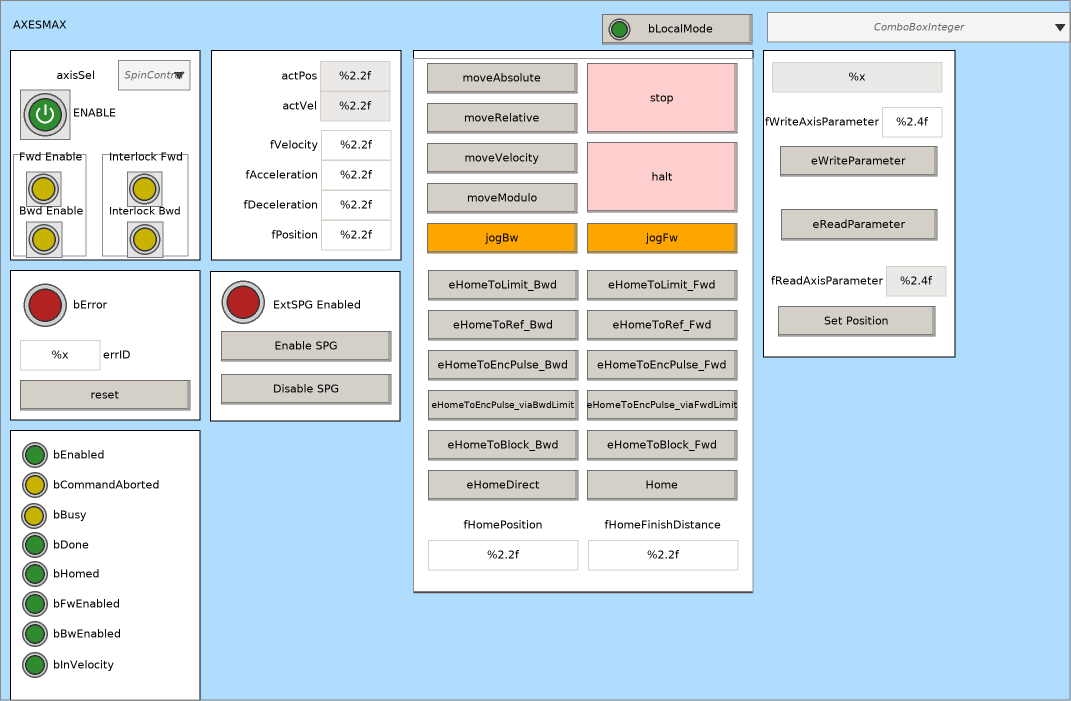
VISUALIZATION MainVisu  // 1071x701
    Rectangle (210,271 190x150)
    Rectangle (413,50 340x542)
    GroupBox (413,50 340x543)
        Button (174,92 150x70), "halt", pressed state: GVL.astAxes[Main.hmiAxisSelection].stControl.bHalt, text list: "languageSupport", text index: "halt"
            toggle GVL.astAxes[Main.hmiAxisSelection].stControl.bHalt
        Button (174,420 150x30), "Home", text list: 'languageSupport', text index: "Home"
            OnMouseClick: execute { GVL.astAxes[Main.hmiAxisSelection].stControl.eCommand:=E_MotionFunctions.eHome; GVL.astAxes[Main.hmiAxisSelection].stControl.bExecute:=TRUE; }
        Button (15,380 150x30), "eHomeToBlock_Bwd", text list: 'languageSupport', text index: "eHomeToBlock_Bwd"
            OnMouseClick: execute {
                GVL.astAxes[Main.hmiAxisSelection].stControl.eCommand:=E_MotionFunctions.eHome;
                GVL.astAxes[Main.hmiAxisSelection].stHomingConfig.eHomeSeq:=E_HomingRoutines.eHomeToBlock_Bwd;
                GVL.astAxes[Main.hmiAxisSelection].stControl.bExecute:=TRUE;
            }
    GroupBox (10,50 190x210)
        Rectangle (0,0 190x210)
        GroupBox (3,96 73x110)
        GroupBox (92,96 86x110)
        Textfield (60,50 92x26), "ENABLE", text list: 'languageSupport', text index: "enable"
        PushSwitchLed (16,118 35x42), variable: GVL.astAxes[MAIN.hmiAxisSelection].stInputs.bLimitFwd, behaviour: TOGGLE, style: Switch-PushSwitchLed-Yellow
        PushSwitchLed (16,170 36x39), variable: GVL.astAxes[MAIN.hmiAxisSelection].stInputs.bLimitBwd, behaviour: TOGGLE, style: Switch-PushSwitchLed-Yellow
        SpinControl (108,10 72x30), variable: MAIN.hmiAxisSelection
            p651134158: GVL_APP.nAXIS_NUM
        Textfield (23,13 86x25), "axisSel", text variable: GVL_APP.nAXIS_NUM, text list: "languageSupport", text index: "axisSel"
        PowerSwitch (10,38 50x53), variable: GVL.astAxes[MAIN.hmiAxisSelection].stControl.bEnable, behaviour: TOGGLE, style: Switch-PowerSwitch-Green
        PushSwitchLed (117,118 35x42), variable: GVL.astAxes[MAIN.hmiAxisSelection].stControl.bInterlockFwd, behaviour: TOGGLE, style: Switch-PushSwitchLed-Yellow
        PushSwitchLed (117,170 36x39), variable: GVL.astAxes[MAIN.hmiAxisSelection].stControl.bInterlockBwd, behaviour: TOGGLE, style: Switch-PushSwitchLed-Yellow
        Textfield (6,94 76x26), "Fwd Enable", text list: 'languageSupport', text index: "enFW"
        Textfield (6,148 76x26), "Bwd Enable", text list: 'languageSupport', text index: "enBW"
        Textfield (96,94 76x26), "Interlock Fwd", text list: 'languageSupport', text index: "bAxisInterlockFwd"
        Textfield (96,148 76x26), "Interlock Bwd", text list: 'languageSupport', text index: "bAxisInterlockBwd"
    Textfield (10,10 231x30), "AXESMAX", text variable: GVL_APP.nAXIS_NUM, text list: "languageSupport", text index: "axesAvailable"
    Button (427,63 150x30), "moveAbsolute", text list: "languageSupport", text index: "moveAbsolute"
        OnMouseClick: execute { GVL.astAxes[MAIN.hmiAxisSelection].stControl.eCommand:=E_MotionFunctions.eMoveAbsolute; GVL.astAxes[MAIN.hmiAxisSelection].stControl.bExecute:=TRUE; }
    Button (427,143 150x30), "moveVelocity", text list: "languageSupport", text index: "moveVelocity"
        OnMouseClick: execute { GVL.astAxes[Main.hmiAxisSelection].stControl.eCommand:=E_MotionFunctions.eMoveVelocity; GVL.astAxes[Main.hmiAxisSelection].stControl.bExecute:=TRUE; }
    Button (427,103 150x30), "moveRelative", text list: "languageSupport", text index: "moveRelative"
        OnMouseClick: execute { GVL.astAxes[Main.hmiAxisSelection].stControl.eCommand:=E_MotionFunctions.eMoveRelative; GVL.astAxes[Main.hmiAxisSelection].stControl.bExecute:=TRUE; }
    Button (427,183 150x30), "moveModulo", text list: "languageSupport", text index: "moveModulo"
        OnMouseClick: execute { GVL.astAxes[Main.hmiAxisSelection].stControl.eCommand:=E_MotionFunctions.eMoveModulo; GVL.astAxes[Main.hmiAxisSelection].stControl.bExecute:=TRUE; }
    Button (587,63 150x70), "stop", pressed state: GVL.astAxes[Main.hmiAxisSelection].stControl.bStop, text list: "languageSupport", text index: "stop"
        toggle GVL.astAxes[Main.hmiAxisSelection].stControl.bStop
    Button (427,223 150x30), "jogBw", text list: "languageSupport", text index: "jogBw"
        OnMouseDown: execute {
            GVL.astAxes[Main.hmiAxisSelection].stControl.eCommand:=E_MotionFunctions.eMoveVelocity;
            GVL.astAxes[Main.hmiAxisSelection].stControl.fVelocity:=-ABS(GVL.astAxes[Main.hmiAxisSelection].stControl.fJogVelocity)
            GVL.astAxes[Main.hmiAxisSelection].stControl.bExecute:= TRUE;
        }
        OnMouseClick: execute {  }
        OnMouseUp: execute { GVL.astAxes[Main.hmiAxisSelection].stControl.bHalt:= TRUE; }
    Button (587,223 150x30), "jogFw", text list: "languageSupport", text index: "jogFw"
        OnMouseDown: execute {
            GVL.astAxes[Main.hmiAxisSelection].stControl.eCommand:=E_MotionFunctions.eMoveVelocity;
            GVL.astAxes[Main.hmiAxisSelection].stControl.fVelocity:=ABS(GVL.astAxes[Main.hmiAxisSelection].stControl.fJogVelocity)
            GVL.astAxes[Main.hmiAxisSelection].stControl.bExecute:= TRUE;
        }
        OnMouseClick: execute {  }
        OnMouseUp: execute { GVL.astAxes[Main.hmiAxisSelection].stControl.bHalt:= TRUE; }
    GroupBox (10,270 190x150)
        Rectangle (0,0 190x150)
        Textfield (90,70 90x30), "errID", text list: "languageSupport", text index: "errID"
        Textfield (10,70 80x30), "%x", text variable: GVL.astAxes[MAIN.hmiAxisSelection].stStatus.nErrorID
        Lamp1 (10,10 50x50), variable: GVL.astAxes[MAIN.hmiAxisSelection].stStatus.bError, style: Lamp-Lamp1-Red
        Textfield (60,20 120x30), "bError", text list: "languageSupport", text index: "bError"
        Button (10,110 170x30), "reset", pressed state: GVL.astAxes[Main.hmiAxisSelection].stControl.bReset, text list: "languageSupport", text index: "reset"
            OnMouseClick: toggle GVL.astAxes[Main.hmiAxisSelection].stControl.bReset
    GroupBox (10,430 190x271)
        Rectangle (0,0 190x270)
        Lamp1 (10,10 30x30), variable: GVL.astAxes[MAIN.hmiAxisSelection].stStatus.bEnabled, style: Lamp-Lamp1-Green
        Textfield (40,10 140x30), "bEnabled", text list: "languageSupport", text index: "bEnabled"
        Lamp1 (10,40 30x30), variable: GVL.astAxes[MAIN.hmiAxisSelection].stStatus.bCommandAborted, style: Lamp-Lamp1-Yellow
        Textfield (40,40 140x30), "bCommandAborted", text list: "languageSupport", text index: "bWarning"
        Textfield (40,70 140x30), "bBusy", text list: "languageSupport", text index: "bBusy"
        Lamp1 (10,100 30x30), variable: GVL.astAxes[MAIN.hmiAxisSelection].stStatus.bDone, style: Lamp-Lamp1-Green
        Textfield (40,100 140x30), "bDone", text list: 'languageSupport', text index: "bDone"
        Lamp1 (10,129 30x30), variable: GVL.astAxes[MAIN.hmiAxisSelection].stStatus.bHomed, style: Lamp-Lamp1-Green
        Textfield (40,129 140x30), "bHomed", text list: "languageSupport", text index: "bHomed"
        Lamp1 (10,159 30x30), variable: GVL.astAxes[MAIN.hmiAxisSelection].stStatus.bFwEnabled AND NOT GVL.astAxes[MAIN.hmiAxisSelection].stStatus.bInterlockedFwd, style: Lamp-Lamp1-Green
        Lamp1 (10,189 30x30), variable: GVL.astAxes[MAIN.hmiAxisSelection].stStatus.bBwEnabled AND NOT GVL.astAxes[MAIN.hmiAxisSelection].stStatus.bInterlockedBwd, style: Lamp-Lamp1-Green
        Textfield (40,159 140x30), "bFwEnabled", text list: "languageSupport", text index: "bFwEnabled"
        Textfield (40,189 140x30), "bBwEnabled", text list: "languageSupport", text index: "bBwEnabled"
        Lamp1 (9,71 30x30), variable: GVL.astAxes[MAIN.hmiAxisSelection].stStatus.bBusy, style: Lamp-Lamp1-Yellow
        Lamp1 (10,220 30x30), variable: GVL.astAxes[MAIN.hmiAxisSelection].stStatus.bInVelocity, style: Lamp-Lamp1-Green
    GroupBox (211,50 190x210)
        Rectangle (0,0 190x210)
        Textfield (10,80 100x30), "fVelocity", text list: "languageSupport", text index: "fVelocity"
        Textfield (110,80 70x30), "%2.2f", text variable: GVL.astAxes[MAIN.hmiAxisSelection].stControl.fVelocity
            OnMouseClick: write the text variable via Default
        Textfield (10,110 100x30), "fAcceleration", text list: "languageSupport", text index: "fAcceleration"
        Textfield (110,110 70x30), "%2.2f", text variable: GVL.astAxes[MAIN.hmiAxisSelection].stControl.fAcceleration
            OnMouseClick: write the text variable via Default
        Textfield (10,140 100x30), "fDeceleration", text list: "languageSupport", text index: "fDeceleration"
        Textfield (110,140 70x30), "%2.2f", text variable: GVL.astAxes[MAIN.hmiAxisSelection].stControl.fDeceleration
            OnMouseClick: write the text variable via Default
        Textfield (10,170 100x30), "fPosition", text list: "languageSupport", text index: "fPosition"
        Textfield (110,170 70x30), "%2.2f", text variable: GVL.astAxes[MAIN.hmiAxisSelection].stControl.fPosition
            OnMouseClick: write the text variable via Default
        Textfield (109,11 70x30), "%2.2f", text variable: GVL.astAxes[MAIN.hmiAxisSelection].stStatus.fActPosition
        Textfield (9,11 100x30), "actPos", text list: "languageSupport", text index: "actposition"
        Textfield (9,41 100x30), "actVel", text list: "languageSupport", text index: "actVelocity"
        Textfield (109,41 70x30), "%2.2f", text variable: GVL.astAxes[MAIN.hmiAxisSelection].stStatus.fActVelocity
    Button (428,310 150x30), "eHomeToRef_Bwd", text list: 'languageSupport', text index: "eHomeToRef_Bwd"
        OnMouseClick: execute {
            GVL.astAxes[Main.hmiAxisSelection].stControl.eCommand:=E_MotionFunctions.eHome;
            GVL.astAxes[Main.hmiAxisSelection].stHomingConfig.eHomeSeq:=E_HomingRoutines.eHomeToRef_Bwd;
            GVL.astAxes[Main.hmiAxisSelection].stControl.bExecute:=TRUE;
        }
    Button (587,310 150x30), "eHomeToRef_Fwd", text list: "languageSupport", text index: "eHomeToRef_Fwd"
        OnMouseClick: execute {
            GVL.astAxes[Main.hmiAxisSelection].stControl.eCommand:=E_MotionFunctions.eHome;
            GVL.astAxes[Main.hmiAxisSelection].stHomingConfig.eHomeSeq:=E_HomingRoutines.eHomeToRef_Fwd;
            GVL.astAxes[Main.hmiAxisSelection].stControl.bExecute:=TRUE;
        }
    Button (428,350 150x30), "eHomeToEncPulse_Bwd", text list: 'languageSupport', text index: "eHomeToEncPulse_Bwd"
        OnMouseClick: execute {
            GVL.astAxes[Main.hmiAxisSelection].stControl.eCommand:=E_MotionFunctions.eHome;
            GVL.astAxes[Main.hmiAxisSelection].stHomingConfig.eHomeSeq:=E_HomingRoutines.eHomeToEncPulse_Bwd;
            GVL.astAxes[Main.hmiAxisSelection].stControl.bExecute:=TRUE;
        }
    Button (587,350 150x30), "eHomeToEncPulse_Fwd", text list: "languageSupport", text index: "eHomeToEncPulse_Fwd"
        OnMouseClick: execute {
            GVL.astAxes[Main.hmiAxisSelection].stControl.eCommand:=E_MotionFunctions.eHome;
            GVL.astAxes[Main.hmiAxisSelection].stHomingConfig.eHomeSeq:=E_HomingRoutines.eHomeToEncPulse_Fwd;
            GVL.astAxes[Main.hmiAxisSelection].stControl.bExecute:=TRUE;
        }
    Button (428,470 150x30), "eHomeDirect", text list: 'languageSupport', text index: "eHomeDirect"
        OnMouseClick: execute {
            GVL.astAxes[Main.hmiAxisSelection].stControl.eCommand:=E_MotionFunctions.eHome;
            GVL.astAxes[Main.hmiAxisSelection].stHomingConfig.eHomeSeq:=E_HomingRoutines.eHomeDirect;
            GVL.astAxes[Main.hmiAxisSelection].stControl.bExecute:=TRUE;
        }
    Button (428,270 150x30), "eHomeToLimit_Bwd", text list: 'languageSupport', text index: "eHomeToLimit_Bwd"
        OnMouseClick: execute {
            GVL.astAxes[Main.hmiAxisSelection].stControl.eCommand:=E_MotionFunctions.eHome;
            GVL.astAxes[Main.hmiAxisSelection].stHomingConfig.eHomeSeq:=E_HomingRoutines.eHomeToLimit_Bwd;
            GVL.astAxes[Main.hmiAxisSelection].stControl.bExecute:=TRUE;
        }
    Button (587,270 150x30), "eHomeToLimit_Fwd", text list: "languageSupport", text index: "eHomeToLimit_Fwd"
        OnMouseClick: execute {
            GVL.astAxes[Main.hmiAxisSelection].stControl.eCommand:=E_MotionFunctions.eHome;
            GVL.astAxes[Main.hmiAxisSelection].stHomingConfig.eHomeSeq:=E_HomingRoutines.eHomeToLimit_Fwd;
            GVL.astAxes[Main.hmiAxisSelection].stControl.bExecute:=TRUE;
        }
    Textfield (428,540 150x30), "%2.2f", text variable: GVL.astAxes[MAIN.hmiAxisSelection].stHomingConfig.fHomePosition
        OnMouseClick: write GVL.astAxes[MAIN.hmiAxisSelection].stHomingConfig.fHomePosition via Default
    Button (428,390 150x30), "eHomeToEncPulse_viaBwdLimit", text list: 'languageSupport', text index: "eHomeToEncPulse_viaBwdLimit"
        OnMouseClick: execute {
            GVL.astAxes[Main.hmiAxisSelection].stControl.eCommand:=E_MotionFunctions.eHome;
            GVL.astAxes[Main.hmiAxisSelection].stHomingConfig.eHomeSeq:=E_HomingRoutines.eHomeToEncPulse_viaBwdLimit;
            GVL.astAxes[Main.hmiAxisSelection].stControl.bExecute:=TRUE;
        }
    Button (587,390 150x30), "eHomeToEncPulse_viaFwdLimit", text list: "languageSupport", text index: "eHomeToEncPulse_viaFwdLimit"
        OnMouseClick: execute {
            GVL.astAxes[Main.hmiAxisSelection].stControl.eCommand:=E_MotionFunctions.eHome;
            GVL.astAxes[Main.hmiAxisSelection].stHomingConfig.eHomeSeq:=E_HomingRoutines.eHomeToEncPulse_viaFwdLimit;
            GVL.astAxes[Main.hmiAxisSelection].stControl.bExecute:=TRUE;
        }
    Textfield (588,540 150x30), "%2.2f", text variable: GVL.astAxes[MAIN.hmiAxisSelection].stHomingConfig.fHomeFinishDistance, text list: ''
        OnMouseClick: write GVL.astAxes[MAIN.hmiAxisSelection].stHomingConfig.fHomeFinishDistance via Default
    Textfield (428,510 150x30), "fHomePosition", text list: "languageSupport", text index: "fHomePosition"
    Textfield (588,510 150x30), "fHomeFinishDistance", text list: "languageSupport", text index: "fHomeFinishDistance"
    Group (602,14 150x30)
        Button (0,0 150x30), "bLocalMode", text list: 'languageSupport', text index: bLocalMode
            OnMouseClick: toggle bLocalMode
        Lamp1 (5,3 25x25), variable: bLocalMode, style: Lamp-Lamp1-Green
    Rectangle (763,50 192x307)
    Button (780,146 157x30), "eWriteParameter", text list: "languageSupport", text index: "eWriteParameter"
        OnMouseClick: execute { GVL.astAxes[MAIN.hmiAxisSelection].stControl.eCommand:=E_MotionFunctions.eWriteParameter; GVL.astAxes[MAIN.hmiAxisSelection].stControl.bExecute:=TRUE; }
    Textfield (772,62 170x30), "%x", text variable: astAxes[MAIN.hmiAxisSelection].stConfig.eAxisParameters
        OnMouseClick: write GVL.astAxes[MAIN.hmiAxisSelection].stConfig.eAxisParameters via Default
    Textfield (762,107 120x30), "fWriteAxisParameter", text list: "languageSupport", text index: "fWriteAxisParameter"
    Textfield (882,107 60x30), "%2.4f", text variable: astAxes[MAIN.hmiAxisSelection].stConfig.fWriteAxisParameter
        OnMouseClick: write GVL.astAxes[MAIN.hmiAxisSelection].stConfig.fWriteAxisParameter via Default
    Textfield (886,266 60x30), "%2.4f", text variable: astAxes[MAIN.hmiAxisSelection].stConfig.fReadAxisParameter
        OnMouseClick: write GVL.astAxes[MAIN.hmiAxisSelection].stConfig.fReadAxisParameter via Default
    Textfield (766,266 120x30), "fReadAxisParameter", text list: "languageSupport", text index: "fReadAxisParameter"
    Button (781,209 156x31), "eReadParameter", text list: 'languageSupport', text index: "eReadParameter"
        OnMouseClick: execute { GVL.astAxes[MAIN.hmiAxisSelection].stControl.eCommand:=E_MotionFunctions.eReadParameter; GVL.astAxes[MAIN.hmiAxisSelection].stControl.bExecute:=TRUE; }
    ComboBoxInteger (767,12 304x30), variable: GVL.astAxes[MAIN.hmiAxisSelection].stConfig.eAxisParameters, text list: 'ParameterTextList'
    Textfield (50,650 140x30), "bInVelocity", text list: 'languageSupport', text index: "bInVelocity"
    Button (587,430 150x30), "eHomeToBlock_Fwd", text list: "languageSupport", text index: "eHomeToBlock_Fwd"
        OnMouseClick: execute {
            GVL.astAxes[Main.hmiAxisSelection].stControl.eCommand:=E_MotionFunctions.eHome;
            GVL.astAxes[Main.hmiAxisSelection].stHomingConfig.eHomeSeq:=E_HomingRoutines.eHomeToBlock_Fwd;
            GVL.astAxes[Main.hmiAxisSelection].stControl.bExecute:=TRUE;
        }
    Textfield (270,290 120x30), "ExtSPG Enabled", text list: "languageSupport", text index: "bError"
    Lamp1 (218,277 50x50), variable: GVL.astAxes[MAIN.hmiAxisSelection].stStatus.SPGEnabled, style: Lamp-Lamp1-Red
    Button (221,331 170x30), "Enable SPG", pressed state: GVL.astAxes[Main.hmiAxisSelection].stControl.bReset, text list: "languageSupport", text index: "reset"
        OnMouseClick: toggle GVL.astAxes[Main.hmiAxisSelection].stSpg.EnableSPG
    Button (221,374 170x30), "Disable SPG", pressed state: GVL.astAxes[Main.hmiAxisSelection].stControl.bReset, text list: "languageSupport", text index: "reset"
        OnMouseClick: toggle GVL.astAxes[Main.hmiAxisSelection].stSpg.DisableSPG
    Button (778,306 157x30), "Set Position", text list: "languageSupport", text index: "eWriteParameter"
        OnMouseClick: execute { GVL.astAxes[MAIN.hmiAxisSelection].stControl.eCommand:=E_MotionFunctions.eSetPosition; GVL.astAxes[MAIN.hmiAxisSelection].stControl.bExecute:=TRUE; }
END_VISUALIZATION

(* stored: Version 1.1.0.1, ProductVersion 3.1.4024.11
   Visu MainVisu: Id {98c8ae72-e756-4d11-b6a5-5914882e2424} *)
